// TIA Portal V18 program export: 0 tag tables, 0 data types, 0 data blocks, 5 code blocks (in call order from the OBs), 0 instance data blocks

ORGANIZATION_BLOCK "Main"   // OB1, FBD, ProgramCycle
TITLE = "Main Program Sweep (Cycle)"
{ S7_Optimized_Access := 'TRUE' }
VERSION : 0.1
// stored: AutoNumber true, IsIECCheckEnabled false, SetENOAutomatically false
   VAR_INPUT
      Initial_Call : Bool;   // Initial call of this OB
      Remanence : Bool;   // =True, if remanent data are available
   END_VAR
   VAR_TEMP
      Diag_Ret_Value1 : Int;
   END_VAR
BEGIN

REGION Network 1: Module State of a PROFINET Dev
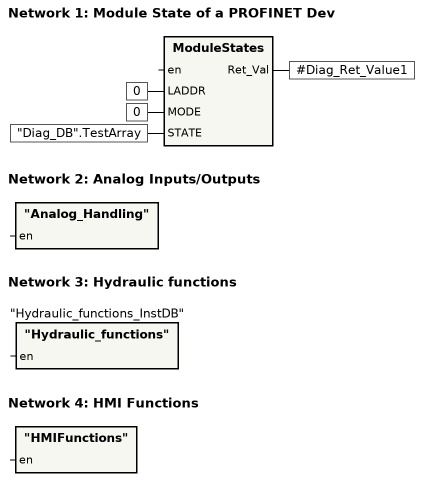
   #Diag_Ret_Value1 := ModuleStates(LADDR := 0, MODE := 0, STATE := "Diag_DB".TestArray);
END_REGION

REGION Network 2: Analog Inputs/Outputs
   "Analog_Handling"();
END_REGION

REGION Network 3: Hydraulic functions
   "Hydraulic_functions_InstDB"();   // "Hydraulic_functions"
END_REGION

REGION Network 4: HMI Functions
   "HMIFunctions"();
END_REGION
END_ORGANIZATION_BLOCK

FUNCTION "Analog_Handling" : Void   // FC3, FBD
TITLE = Analog Handling
{ S7_Optimized_Access := 'TRUE' }
VERSION : 0.1
// stored: AutoNumber true, IsIECCheckEnabled false, SetENOAutomatically false, UDAEnableTagReadback false
   VAR_TEMP
      Dummy11 : Bool;
      Dummy21 : Bool;
   END_VAR
BEGIN

REGION Network 1: **************INPUTS*************
END_REGION

REGION Network 2 (SCL): SCL Network
   IF #Dummy1 THEN
       #Dummy2 := FALSE;    // Statement section IF

   END_IF;
END_REGION

REGION Network 3: CI Proportional Valve Input
   // Rexroth Bef Prop Valve
   // IN: 0-27648
   // UT: 0-100
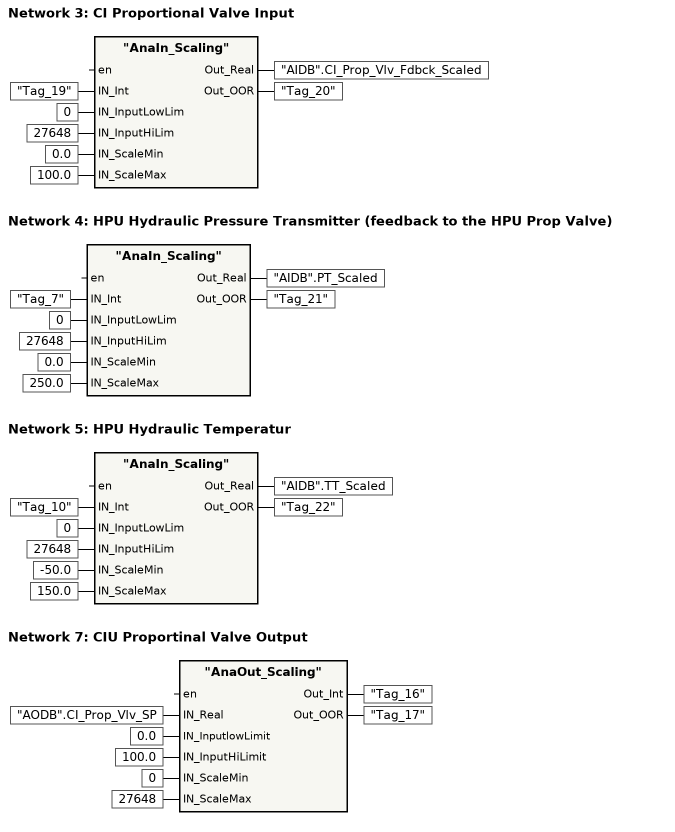
   "AnaIn_Scaling"(IN_Int := "Tag_19",
                   IN_InputLowLim := 0,
                   IN_InputHiLim := 27648,
                   IN_ScaleMin := 0.0,
                   IN_ScaleMax := 100.0,
                   Out_Real => "AIDB".CI_Prop_Vlv_Fdbck_Scaled,
                   Out_OOR => "Tag_20");
END_REGION

REGION Network 4: HPU Hydraulic Pressure Transmitter (feedback to the HPU Prop Valve)
   // IFM PT5401
   // 0-250 bar/4-20mA
   "AnaIn_Scaling"(IN_Int := "Tag_7",
                   IN_InputLowLim := 0,
                   IN_InputHiLim := 27648,
                   IN_ScaleMin := 0.0,
                   IN_ScaleMax := 250.0,
                   Out_Real => "AIDB".PT_Scaled,
                   Out_OOR => "Tag_21");
END_REGION

REGION Network 5: HPU Hydraulic Temperatur
   // IFM TN2435
   // -50...150 grader /4-20mA
   "AnaIn_Scaling"(IN_Int := "Tag_10",
                   IN_InputLowLim := 0,
                   IN_InputHiLim := 27648,
                   IN_ScaleMin := -50.0,
                   IN_ScaleMax := 150.0,
                   Out_Real => "AIDB".TT_Scaled,
                   Out_OOR => "Tag_22");
END_REGION

REGION Network 6: **************OUTPUTS**************
END_REGION

REGION Network 7: CIU Proportinal Valve Output
   "AnaOut_Scaling"(IN_Real := "AODB".CI_Prop_Vlv_SP,
                    IN_InputlowLimit := 0.0,
                    IN_InputHiLimit := 100.0,
                    IN_ScaleMin := 0,
                    IN_ScaleMax := 27648,
                    Out_Int => "Tag_16",
                    Out_OOR => "Tag_17");
END_REGION
END_FUNCTION

FUNCTION "AnaIn_Scaling" : Void   // FC5, FBD
TITLE = Analog Scaling of an Input
{ S7_Optimized_Access := 'TRUE' }
VERSION : 0.1
// -Normalize
// -Scale
// -OOR
// stored: AutoNumber true, IsIECCheckEnabled false, SetENOAutomatically false, UDAEnableTagReadback false
   VAR_INPUT
      IN_Int : DInt;   // Sensor Input Val usually PIWxxx
      IN_InputLowLim : Int;   // Min in from PIW sensor usually 0
      IN_InputHiLim : Int;   // Max in from PIW sensor usually 27648
      IN_ScaleMin : Real;   // Min value for the output scaling
      IN_ScaleMax : Real;   // Max value for the output scaling
   END_VAR
   VAR_OUTPUT
      Out_Real : Real;   // Scaled value
      Out_OOR : Bool;   // Out of Range
   END_VAR
   VAR_TEMP
      Out_norm : Real;
      Out_Scaled : Real;
      Dummy1 : Bool;
      Dummy2 : Bool;
   END_VAR
BEGIN

REGION Network 2 (SCL)
   IF #Dummy1 THEN
       #Dummy2 := FALSE;// Statement section IF

   END_IF;
END_REGION

REGION Network 3: HPU Proportional Valve: Normalize & Scaling of Input Feedback [+/-10V]
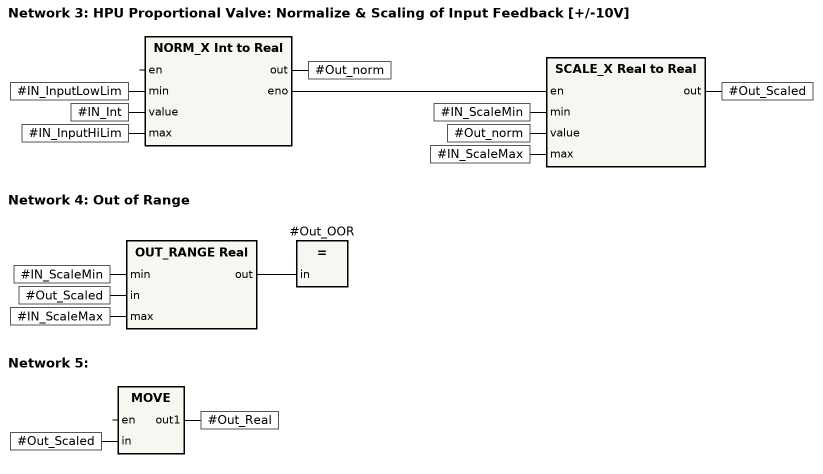
   #Out_norm := NORM_X(MIN := #IN_InputLowLim, VALUE := #IN_Int, MAX := #IN_InputHiLim);
   #Out_Scaled := SCALE_X(MIN := #IN_ScaleMin, VALUE := #Out_norm, MAX := #IN_ScaleMax);
END_REGION

REGION Network 4: Out of Range
   #Out_OOR := (#Out_Scaled < #IN_ScaleMin) OR (#Out_Scaled > #IN_ScaleMax);
END_REGION

REGION Network 5
   #Out_Real := #Out_Scaled;
END_REGION
END_FUNCTION

FUNCTION_BLOCK "Analog_Valve"   // FB104, FBD
TITLE = Analog Valve Control
{ S7_Optimized_Access := 'FALSE' }
AUTHOR : THE
FAMILY : MAIN
NAME : PVALVE
VERSION : 1.1
// stored: AutoNumber false, IsIECCheckEnabled false, SetENOAutomatically false, UDAEnableTagReadback false
   VAR_INPUT
      IN_Em_Stop : Bool;   // Emergency stop / 1=OK, 0=Not OK
      IN_Interlock : Bool;   // Interlock when valve in auto mode / 0=OK, 1=Interlocked
      IN_Reset : Bool;   // Reset alarm / Cmd: Reset
      IN_ValveSP : Real;   // Cmd: Setpoint 0-100%
      IN_ValveSP_Min : Real;   // Min value of the Input Setpoint
      IN_ValveSP_Max : Real;   // Max value of the Iinput setpoint
      IN_Valve_Feedback : Real;   // Sts: Valve feedback 0-100%
      IN_TimerSetpointNotReached : Timer;   // Open % / Close time for valve (sec) / Timer number Setpoint Not Reached
      IN_TimerNotClosing : Timer;   // Timer number Not closing
      IN_TimeoutTime1 : S5Time;   // Real Feedback from Valve / Timeout time in Sec
      IN_TimeoutTime2 : S5Time;   // Timeout time in Sec
   END_VAR
   VAR_OUTPUT
      OUT_ValveSP : Real;   // Setpoint 0-100% Output
      OUT_Valve_Feedback : Real;   // Sts_Valve Feedback 0-100%
      OUT_Valve_Closed : Bool;   // Status: Valve Closed / Sts: Valve closed 1=Closed,0=open
      OUT_Valve_Not_Closing : Bool;   // Alarm: valve not closing / Sts: Timeout Valve Closing
      OUT_SP_Not_Reached : Bool;   // Sts: Setpoint not Reached
      OUT_ValveSP_OOR : Bool;   // Setpoint Value Out Of Range
   END_VAR
   VAR DB_SPECIFIC
      Valve_SP : Real;
      Pos_Deviation_Valve : Real;
      Neg_Deviation_Valve : Real;
      Open_Cmd : Bool;
      Operate : Bool;
   END_VAR
   VAR_TEMP
      SP_Overrange : Bool;
      SP_Underrange : Bool;
   END_VAR
   VAR_TEMP   // added for the SCL form of the ladder/FBD networks
      _w1 : Bool;
      _s5time1 : S5Time;
   END_VAR
BEGIN

REGION Network 1: Internal operate flag
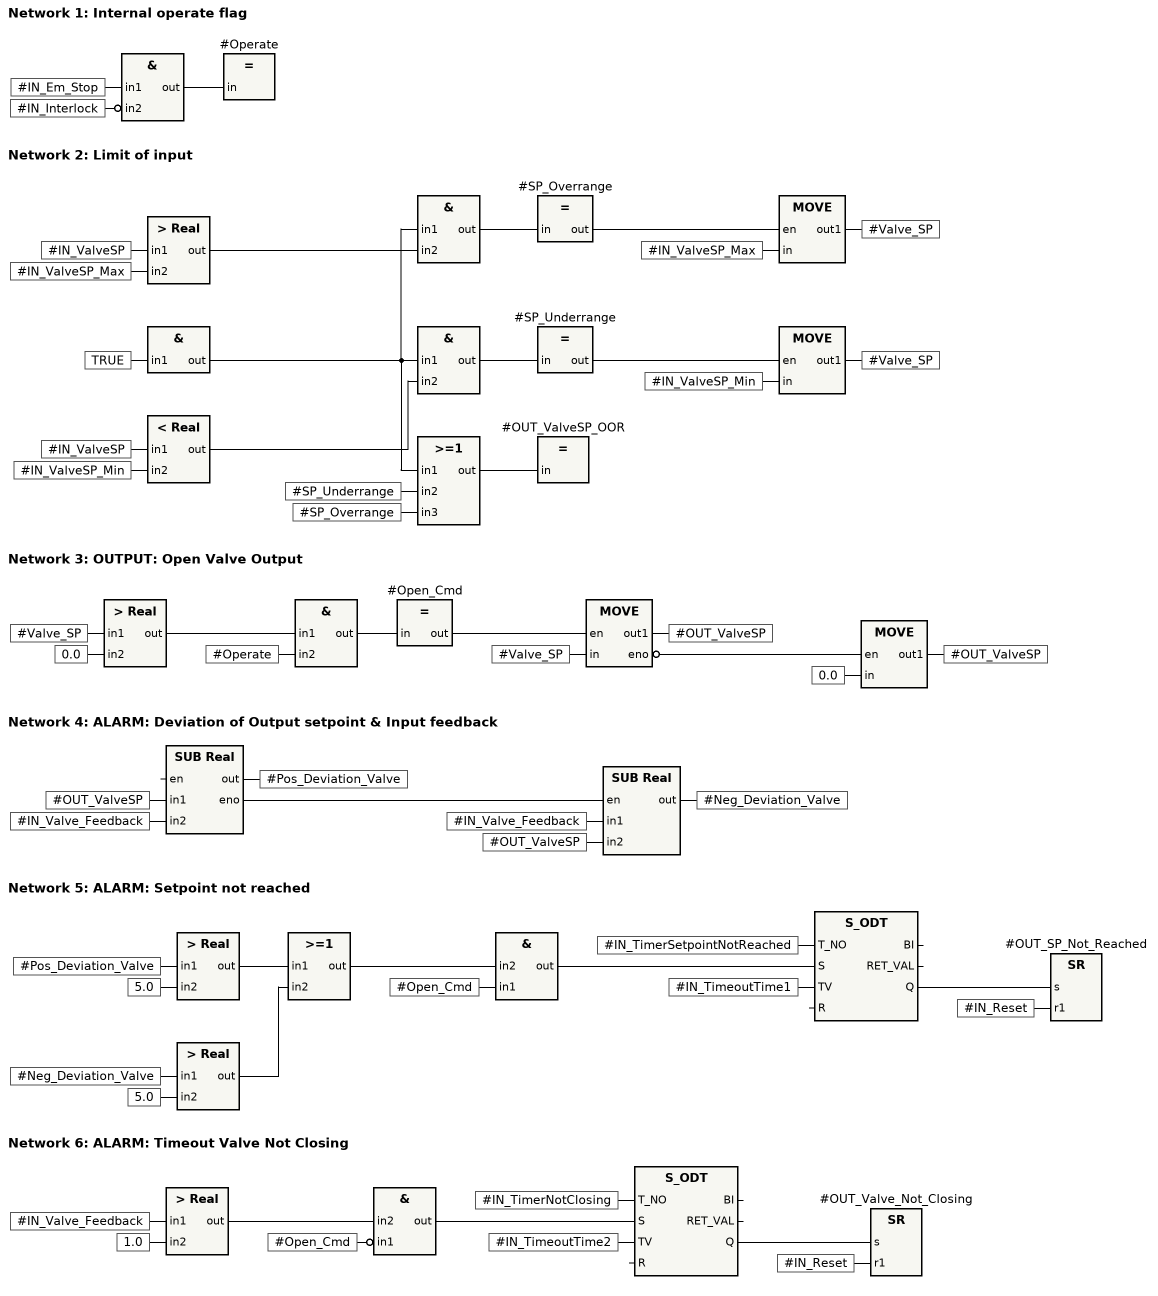
   #Operate := #IN_Em_Stop AND NOT #IN_Interlock;
END_REGION

REGION Network 2: Limit of input
   #SP_Overrange := TRUE AND (#IN_ValveSP > #IN_ValveSP_Max);
   IF #SP_Overrange THEN #Valve_SP := #IN_ValveSP_Max; END_IF;
   #SP_Underrange := TRUE AND (#IN_ValveSP < #IN_ValveSP_Min);
   IF #SP_Underrange THEN #Valve_SP := #IN_ValveSP_Min; END_IF;
   #OUT_ValveSP_OOR := TRUE OR #SP_Underrange OR #SP_Overrange;
END_REGION

REGION Network 3: OUTPUT: Open Valve Output
   #Open_Cmd := (#Valve_SP > 0.0) AND #Operate;
   IF #Open_Cmd THEN #OUT_ValveSP := #Valve_SP; END_IF;
   IF NOT #Open_Cmd THEN #OUT_ValveSP := 0.0; END_IF;
END_REGION

REGION Network 4: ALARM: Deviation of Output setpoint & Input feedback
   // Check if deviation between Output & Fedback
   // ENO of a box is taken as its EN; it also drops when the box reports an error
   #Pos_Deviation_Valve := #OUT_ValveSP - #IN_Valve_Feedback;
   #Neg_Deviation_Valve := #IN_Valve_Feedback - #OUT_ValveSP;
END_REGION

REGION Network 5: ALARM: Setpoint not reached
   #_s5time1 := S_ODT(T_NO := #IN_TimerSetpointNotReached,
                      S := ((#Pos_Deviation_Valve > 5.0) OR (#Neg_Deviation_Valve > 5.0)) AND #Open_Cmd,
                      TV := #IN_TimeoutTime1,
                      Q => #_w1);
   IF #_w1 THEN
       #OUT_SP_Not_Reached := TRUE;   // SR flip-flop
   END_IF;
   IF #IN_Reset THEN #OUT_SP_Not_Reached := FALSE; END_IF;
END_REGION

REGION Network 6: ALARM: Timeout Valve Not Closing
   #_s5time1 := S_ODT(T_NO := #IN_TimerNotClosing,
                      S := (#IN_Valve_Feedback > 1.0) AND NOT #Open_Cmd,
                      TV := #IN_TimeoutTime2,
                      Q => #_w1);
   IF #_w1 THEN
       #OUT_Valve_Not_Closing := TRUE;   // SR flip-flop
   END_IF;
   IF #IN_Reset THEN #OUT_Valve_Not_Closing := FALSE; END_IF;
END_REGION

REGION Network 7: OUTPUT: Valve Feedback to Output
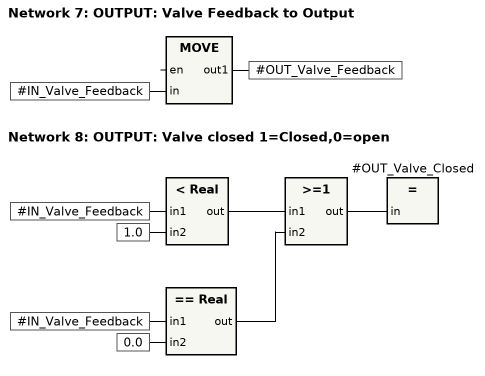
   #OUT_Valve_Feedback := #IN_Valve_Feedback;
END_REGION

REGION Network 8: OUTPUT: Valve closed 1=Closed,0=open
   #OUT_Valve_Closed := (#IN_Valve_Feedback < 1.0) OR (#IN_Valve_Feedback = 0.0);
END_REGION
END_FUNCTION_BLOCK

FUNCTION_BLOCK "B16_TO_W"
{ S7_Optimized_Access := 'TRUE' }
VERSION : 0.4
   VAR_INPUT 
      B_0 : Bool;
      B_1 : Bool;
      B_2 : Bool;
      B_3 : Bool;
      B_4 : Bool;
      B_5 : Bool;
      B_6 : Bool;
      B_7 : Bool;
      B_8 : Bool;
      B_9 : Bool;
      B_10 : Bool;
      B_11 : Bool;
      B_12 : Bool;
      B_13 : Bool;
      B_14 : Bool;
      B_15 : Bool;
   END_VAR

   VAR_OUTPUT 
      OUT_W : Word;
   END_VAR


BEGIN
	#OUT_W.%X0:=#B_0;
	#OUT_W.%X1:=#B_1;
	#OUT_W.%X2:=#B_2;
	#OUT_W.%X3:=#B_3;
	#OUT_W.%X4:=#B_4;
	#OUT_W.%X5:=#B_5;
	#OUT_W.%X6:=#B_6;
	#OUT_W.%X7:=#B_7;
	#OUT_W.%X8:=#B_8;
	#OUT_W.%X9:=#B_9;
	#OUT_W.%X10:=#B_10;
	#OUT_W.%X11:=#B_11;
	#OUT_W.%X12:=#B_12;
	#OUT_W.%X13:=#B_13;
	#OUT_W.%X14:=#B_14;
	#OUT_W.%X15:=#B_15;
	
END_FUNCTION_BLOCK
